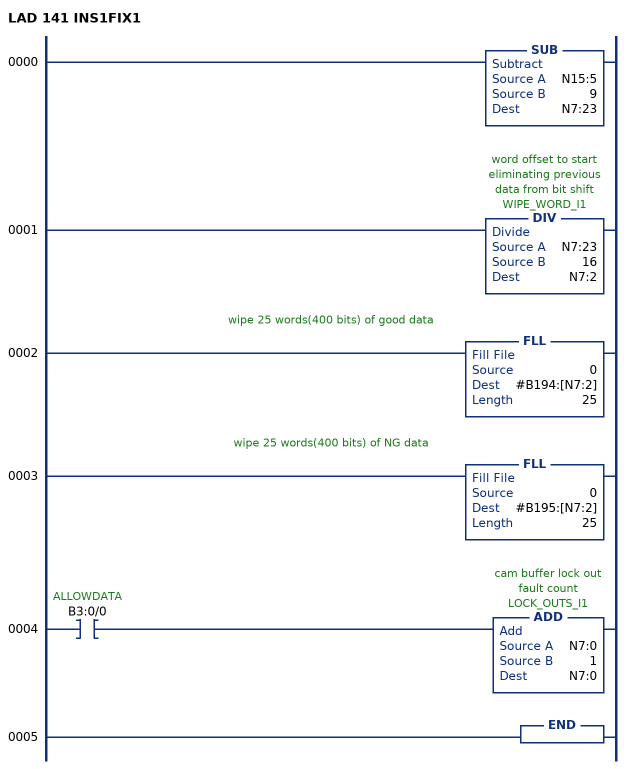
% Rung: 0 %
SOR SUB N15:5 9 N7:23 EOR
%   N15:5  INS_1_TRIG_LOC %
% Rung: 1 %
SOR DIV N7:23 16 N7:2 EOR
%   N7:2  WIPE_WORD_I1  "word offset to start eliminating previous data from bit shift" %
% Rung: 2 %
% wipe 25 words(400 bits) of good data %
SOR FLL 0 #B194:[N7:2] 25 EOR
%   N7:2  WIPE_WORD_I1  "word offset to start eliminating previous data from bit shift" %
% Rung: 3 %
% wipe 25 words(400 bits) of NG data %
SOR FLL 0 #B195:[N7:2] 25 EOR
%   N7:2  WIPE_WORD_I1  "word offset to start eliminating previous data from bit shift" %
% Rung: 4 %
SOR XIC B3:0/0 ADD N7:0 1 N7:0 EOR
%   B3:0/0  ALLOWDATA %
%   N7:0  LOCK_OUTS_I1  "cam buffer lock out fault count" %
% Rung: 5 %
SOR END EOR

LADDER 142 "INS1FIX2"
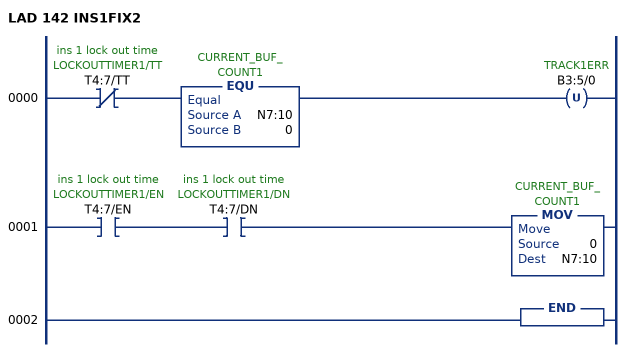
% Rung: 0 %
SOR XIO T4:7/TT EQU N7:10 0 OTU B3:5/0 EOR
%   T4:7  LOCKOUTTIMER1  "ins 1 lock out time" %
%   N7:10  CURRENT_BUF_COUNT1 %
%   B3:5/0  TRACK1ERR %
% Rung: 1 %
SOR XIC T4:7/EN XIC T4:7/DN MOV 0 N7:10 EOR
%   T4:7  LOCKOUTTIMER1  "ins 1 lock out time" %
%   N7:10  CURRENT_BUF_COUNT1 %
% Rung: 2 %
SOR END EOR

LADDER 145 "INS2"
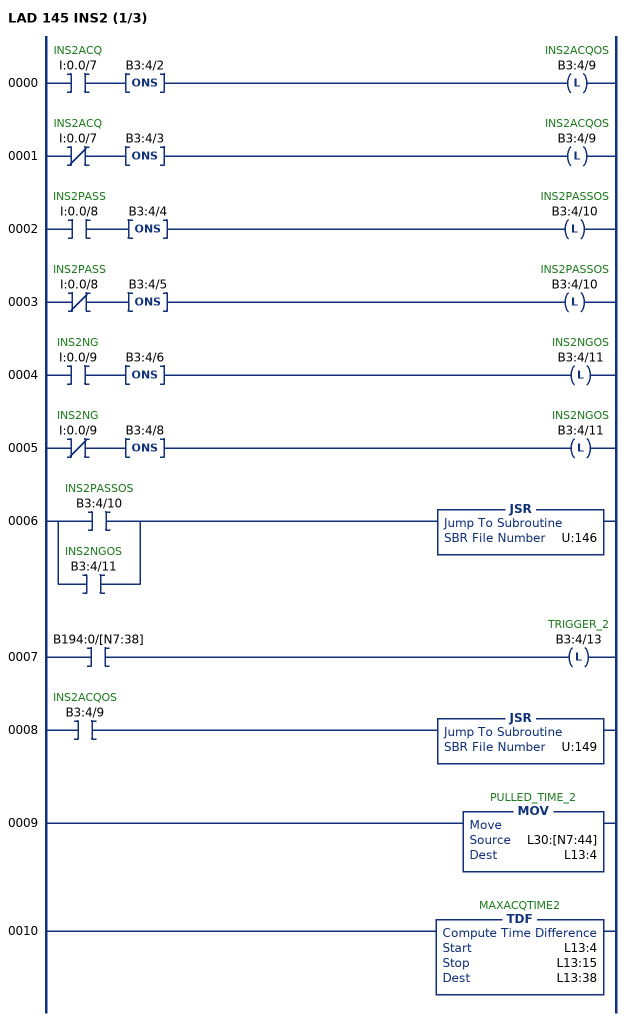
% Rung: 0 %
SOR XIC I:0.0/7 ONS B3:4/2 OTL B3:4/9 EOR
%   I:0.0/7  INS2ACQ %
%   B3:4/9  INS2ACQOS %
% Rung: 1 %
SOR XIO I:0.0/7 ONS B3:4/3 OTL B3:4/9 EOR
%   I:0.0/7  INS2ACQ %
%   B3:4/9  INS2ACQOS %
% Rung: 2 %
SOR XIC I:0.0/8 ONS B3:4/4 OTL B3:4/10 EOR
%   I:0.0/8  INS2PASS %
%   B3:4/10  INS2PASSOS %
% Rung: 3 %
SOR XIO I:0.0/8 ONS B3:4/5 OTL B3:4/10 EOR
%   I:0.0/8  INS2PASS %
%   B3:4/10  INS2PASSOS %
% Rung: 4 %
SOR XIC I:0.0/9 ONS B3:4/6 OTL B3:4/11 EOR
%   I:0.0/9  INS2NG %
%   B3:4/11  INS2NGOS %
% Rung: 5 %
SOR XIO I:0.0/9 ONS B3:4/8 OTL B3:4/11 EOR
%   I:0.0/9  INS2NG %
%   B3:4/11  INS2NGOS %
% Rung: 6 %
SOR BST XIC B3:4/10 NXB XIC B3:4/11 BND JSR U:146 EOR
%   B3:4/10  INS2PASSOS %
%   B3:4/11  INS2NGOS %
% Rung: 7 %
SOR XIC B194:0/[N7:38] OTL B3:4/13 EOR
%   B194:0  BOT_GOOD_FILE %
%   N7:38  INS_2_TRIG_LOC %
%   B3:4/13  TRIGGER_2 %
% Rung: 8 %
SOR XIC B3:4/9 JSR U:149 EOR
%   B3:4/9  INS2ACQOS %
% Rung: 9 %
SOR MOV L30:[N7:44] L13:4 EOR
%   N7:44  OLDEST_PART_INDEX2 %
%   L13:4  PULLED_TIME_2 %
% Rung: 10 %
SOR TDF L13:4 L13:15 L13:38 EOR
%   L13:4  PULLED_TIME_2 %
%   L13:15  BOT_TIME %
%   L13:38  MAXACQTIME2 %

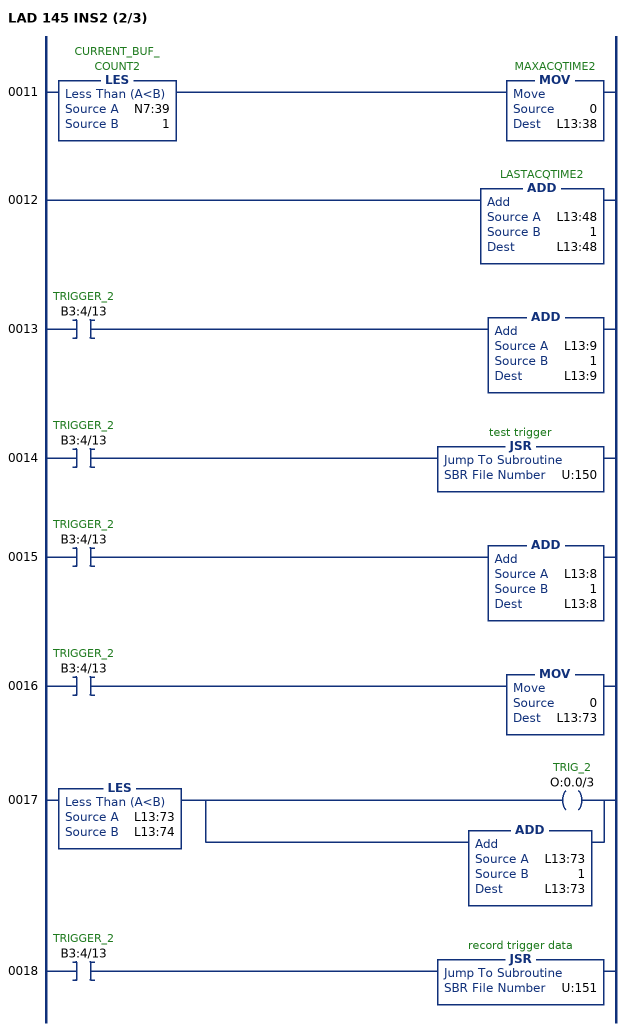
% Rung: 11 %
SOR LES N7:39 1 MOV 0 L13:38 EOR
%   N7:39  CURRENT_BUF_COUNT2 %
%   L13:38  MAXACQTIME2 %
% Rung: 12 %
SOR ADD L13:48 1 L13:48 EOR
%   L13:48  LASTACQTIME2 %
% Rung: 13 %
SOR XIC B3:4/13 ADD L13:9 1 L13:9 EOR
%   B3:4/13  TRIGGER_2 %
% Rung: 14 %
SOR XIC B3:4/13 JSR U:150 EOR
%   B3:4/13  TRIGGER_2 %
%   U:150  "test trigger" %
% Rung: 15 %
SOR XIC B3:4/13 ADD L13:8 1 L13:8 EOR
%   B3:4/13  TRIGGER_2 %
% Rung: 16 %
SOR XIC B3:4/13 MOV 0 L13:73 EOR
%   B3:4/13  TRIGGER_2 %
% Rung: 17 %
SOR LES L13:73 L13:74 BST OTE O:0.0/3 NXB ADD L13:73 1 L13:73 BND EOR
%   O:0.0/3  TRIG_2 %
% Rung: 18 %
SOR XIC B3:4/13 JSR U:151 EOR
%   B3:4/13  TRIGGER_2 %
%   U:151  "record trigger data" %

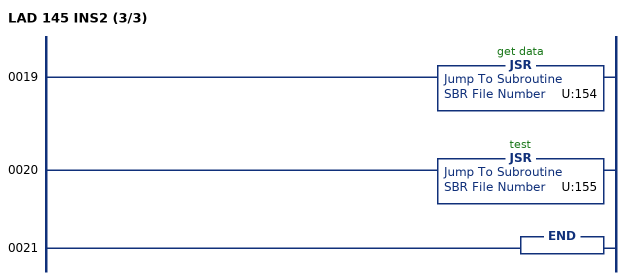
% Rung: 19 %
SOR JSR U:154 EOR
%   U:154  "get data" %
% Rung: 20 %
SOR JSR U:155 EOR
%   U:155  "test" %
% Rung: 21 %
SOR END EOR

LADDER 146 "INS2RESULT"
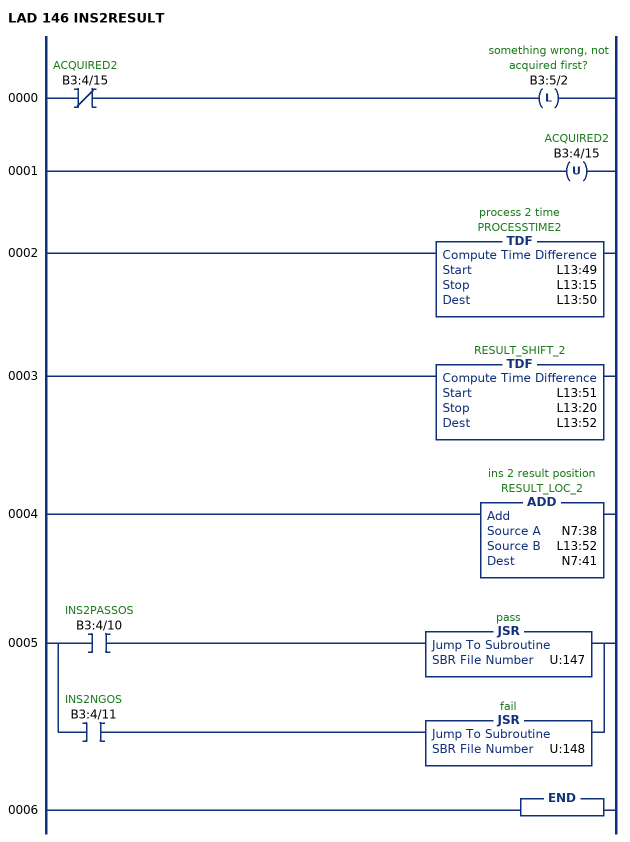
% Rung: 0 %
SOR XIO B3:4/15 OTL B3:5/2 EOR
%   B3:4/15  ACQUIRED2 %
%   B3:5/2  "something wrong, not acquired first?" %
% Rung: 1 %
SOR OTU B3:4/15 EOR
%   B3:4/15  ACQUIRED2 %
% Rung: 2 %
SOR TDF L13:49 L13:15 L13:50 EOR
%   L13:49  TIMEOFACQ2  "the time of the last acquire" %
%   L13:15  BOT_TIME %
%   L13:50  PROCESSTIME2  "process 2 time" %
% Rung: 3 %
SOR TDF L13:51 L13:20 L13:52 EOR
%   L13:51  PROCESS_START_POS_2 %
%   L13:20  BOT_POSITION %
%   L13:52  RESULT_SHIFT_2 %
% Rung: 4 %
SOR ADD N7:38 L13:52 N7:41 EOR
%   N7:38  INS_2_TRIG_LOC %
%   L13:52  RESULT_SHIFT_2 %
%   N7:41  RESULT_LOC_2  "ins 2 result position" %
% Rung: 5 %
SOR BST XIC B3:4/10 JSR U:147 NXB XIC B3:4/11 JSR U:148 BND EOR
%   B3:4/10  INS2PASSOS %
%   U:147  "pass" %
%   B3:4/11  INS2NGOS %
%   U:148  "fail" %
% Rung: 6 %
SOR END EOR

LADDER 147 "INS2PASS"
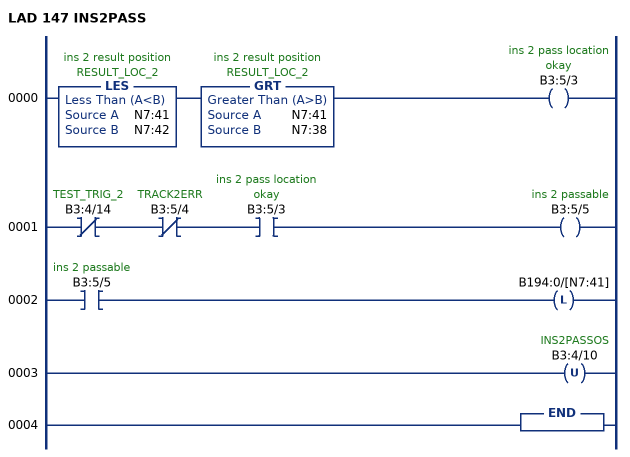
% Rung: 0 %
SOR LES N7:41 N7:42 GRT N7:41 N7:38 OTE B3:5/3 EOR
%   N7:41  RESULT_LOC_2  "ins 2 result position" %
%   N7:42  MAXRSTLOC2 %
%   N7:38  INS_2_TRIG_LOC %
%   B3:5/3  "ins 2 pass location okay" %
% Rung: 1 %
SOR XIO B3:4/14 XIO B3:5/4 XIC B3:5/3 OTE B3:5/5 EOR
%   B3:4/14  TEST_TRIG_2 %
%   B3:5/4  TRACK2ERR %
%   B3:5/3  "ins 2 pass location okay" %
%   B3:5/5  "ins 2 passable" %
% Rung: 2 %
SOR XIC B3:5/5 OTL B194:0/[N7:41] EOR
%   B3:5/5  "ins 2 passable" %
%   B194:0  BOT_GOOD_FILE %
%   N7:41  RESULT_LOC_2  "ins 2 result position" %
% Rung: 3 %
SOR OTU B3:4/10 EOR
%   B3:4/10  INS2PASSOS %
% Rung: 4 %
SOR END EOR

LADDER 148 "INS2FAIL"
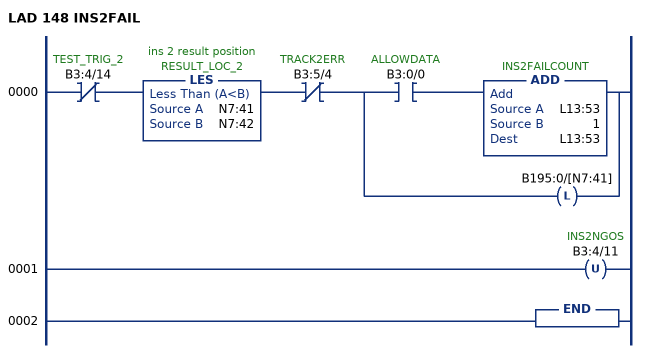
% Rung: 0 %
SOR XIO B3:4/14 LES N7:41 N7:42 XIO B3:5/4 BST XIC B3:0/0 ADD L13:53 1 L13:53 NXB OTL B195:0/[N7:41] BND EOR
%   B3:4/14  TEST_TRIG_2 %
%   N7:41  RESULT_LOC_2  "ins 2 result position" %
%   N7:42  MAXRSTLOC2 %
%   B3:5/4  TRACK2ERR %
%   B3:0/0  ALLOWDATA %
%   L13:53  INS2FAILCOUNT %
%   B195:0  BOT_NG_FILE %
% Rung: 1 %
SOR OTU B3:4/11 EOR
%   B3:4/11  INS2NGOS %
% Rung: 2 %
SOR END EOR

LADDER 149 "INS2ACQ"
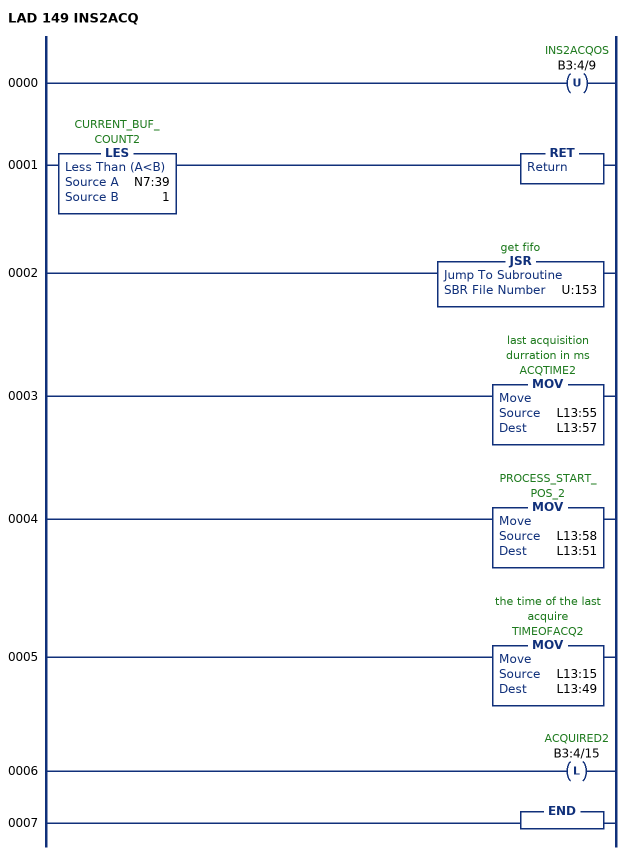
% Rung: 0 %
SOR OTU B3:4/9 EOR
%   B3:4/9  INS2ACQOS %
% Rung: 1 %
SOR LES N7:39 1 RET EOR
%   N7:39  CURRENT_BUF_COUNT2 %
% Rung: 2 %
SOR JSR U:153 EOR
%   U:153  "get fifo" %
% Rung: 3 %
SOR MOV L13:55 L13:57 EOR
%   L13:55  TIME_SPAN2 %
%   L13:57  ACQTIME2  "last acquisition durration in ms" %
% Rung: 4 %
SOR MOV L13:58 L13:51 EOR
%   L13:58  PULLED_POSITION2 %
%   L13:51  PROCESS_START_POS_2 %
% Rung: 5 %
SOR MOV L13:15 L13:49 EOR
%   L13:15  BOT_TIME %
%   L13:49  TIMEOFACQ2  "the time of the last acquire" %
% Rung: 6 %
SOR OTL B3:4/15 EOR
%   B3:4/15  ACQUIRED2 %
% Rung: 7 %
SOR END EOR

LADDER 150 "Q2TIMETEST"
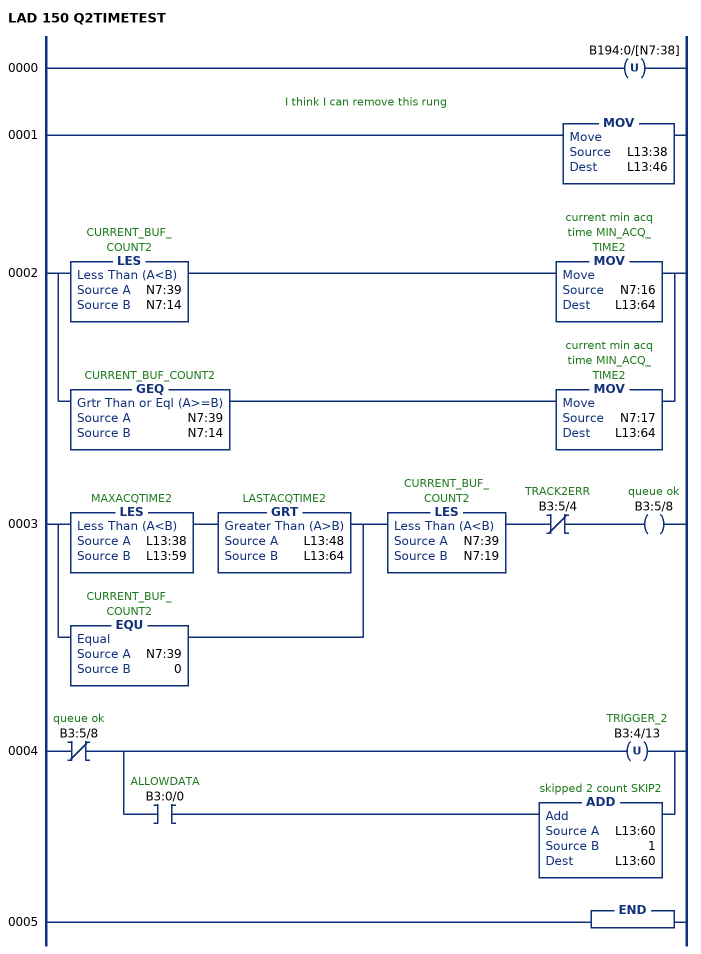
% Rung: 0 %
SOR OTU B194:0/[N7:38] EOR
%   B194:0  BOT_GOOD_FILE %
%   N7:38  INS_2_TRIG_LOC %
% Rung: 1 %
% I think I can remove this rung %
SOR MOV L13:38 L13:46 EOR
%   L13:38  MAXACQTIME2 %
% Rung: 2 %
SOR BST LES N7:39 N7:14 MOV N7:16 L13:64 NXB GEQ N7:39 N7:14 MOV N7:17 L13:64 BND EOR
%   N7:39  CURRENT_BUF_COUNT2 %
%   N7:14  "Max high speed buffers" %
%   N7:16  "high speed acquisition time" %
%   L13:64  MIN_ACQ_TIME2  "current min acq time" %
%   N7:17  "low speed acquisition time" %
% Rung: 3 %
SOR BST LES L13:38 L13:59 GRT L13:48 L13:64 NXB EQU N7:39 0 BND LES N7:39 N7:19 XIO B3:5/4 OTE B3:5/8 EOR
%   L13:38  MAXACQTIME2 %
%   L13:59  ACQTIMELIMIT2 %
%   L13:48  LASTACQTIME2 %
%   L13:64  MIN_ACQ_TIME2  "current min acq time" %
%   N7:39  CURRENT_BUF_COUNT2 %
%   N7:19  MAX_BUFF  "maximum buffers" %
%   B3:5/4  TRACK2ERR %
%   B3:5/8  "queue ok" %
% Rung: 4 %
SOR XIO B3:5/8 BST OTU B3:4/13 NXB XIC B3:0/0 ADD L13:60 1 L13:60 BND EOR
%   B3:5/8  "queue ok" %
%   B3:4/13  TRIGGER_2 %
%   B3:0/0  ALLOWDATA %
%   L13:60  SKIP2  "skipped 2 count" %
% Rung: 5 %
SOR END EOR

LADDER 151 "INS2TRIG"
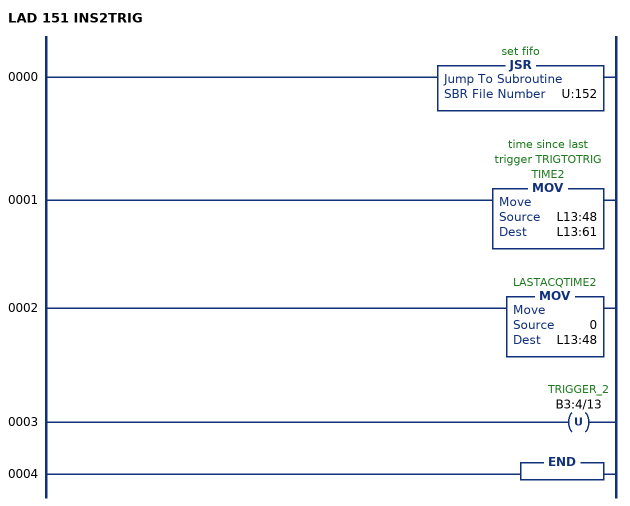
% Rung: 0 %
SOR JSR U:152 EOR
%   U:152  "set fifo" %
% Rung: 1 %
SOR MOV L13:48 L13:61 EOR
%   L13:48  LASTACQTIME2 %
%   L13:61  TRIGTOTRIGTIME2  "time since last trigger" %
% Rung: 2 %
SOR MOV 0 L13:48 EOR
%   L13:48  LASTACQTIME2 %
% Rung: 3 %
SOR OTU B3:4/13 EOR
%   B3:4/13  TRIGGER_2 %
% Rung: 4 %
SOR END EOR

LADDER 152 "FIFO2SET"
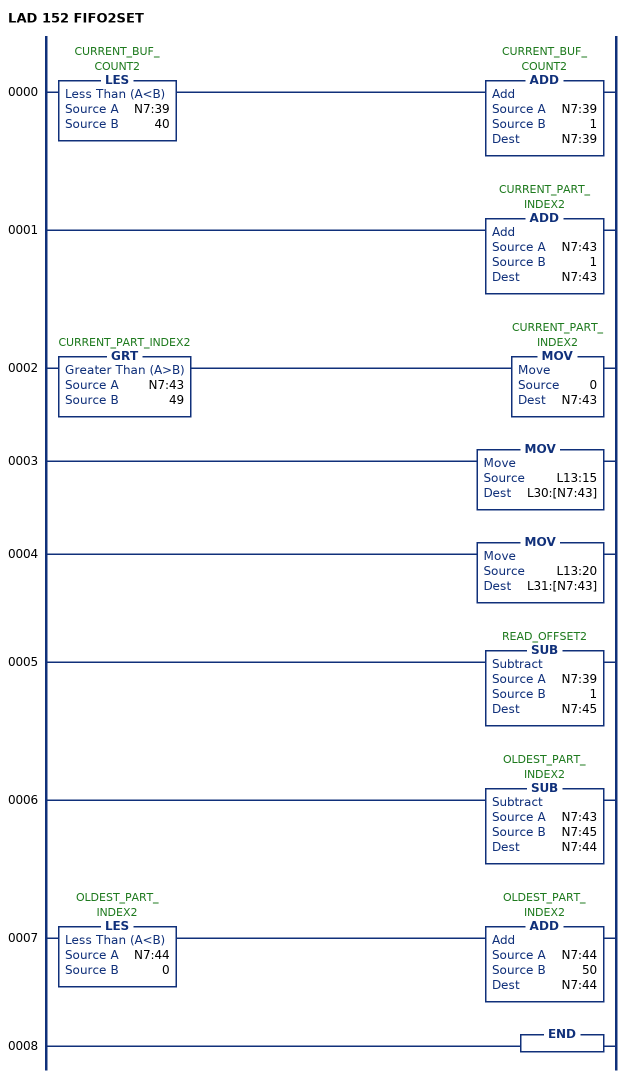
% Rung: 0 %
SOR LES N7:39 40 ADD N7:39 1 N7:39 EOR
%   N7:39  CURRENT_BUF_COUNT2 %
% Rung: 1 %
SOR ADD N7:43 1 N7:43 EOR
%   N7:43  CURRENT_PART_INDEX2 %
% Rung: 2 %
SOR GRT N7:43 49 MOV 0 N7:43 EOR
%   N7:43  CURRENT_PART_INDEX2 %
% Rung: 3 %
SOR MOV L13:15 L30:[N7:43] EOR
%   L13:15  BOT_TIME %
%   N7:43  CURRENT_PART_INDEX2 %
% Rung: 4 %
SOR MOV L13:20 L31:[N7:43] EOR
%   L13:20  BOT_POSITION %
%   N7:43  CURRENT_PART_INDEX2 %
% Rung: 5 %
SOR SUB N7:39 1 N7:45 EOR
%   N7:39  CURRENT_BUF_COUNT2 %
%   N7:45  READ_OFFSET2 %
% Rung: 6 %
SOR SUB N7:43 N7:45 N7:44 EOR
%   N7:43  CURRENT_PART_INDEX2 %
%   N7:45  READ_OFFSET2 %
%   N7:44  OLDEST_PART_INDEX2 %
% Rung: 7 %
SOR LES N7:44 0 ADD N7:44 50 N7:44 EOR
%   N7:44  OLDEST_PART_INDEX2 %
% Rung: 8 %
SOR END EOR

LADDER 153 "FIFO2GET"
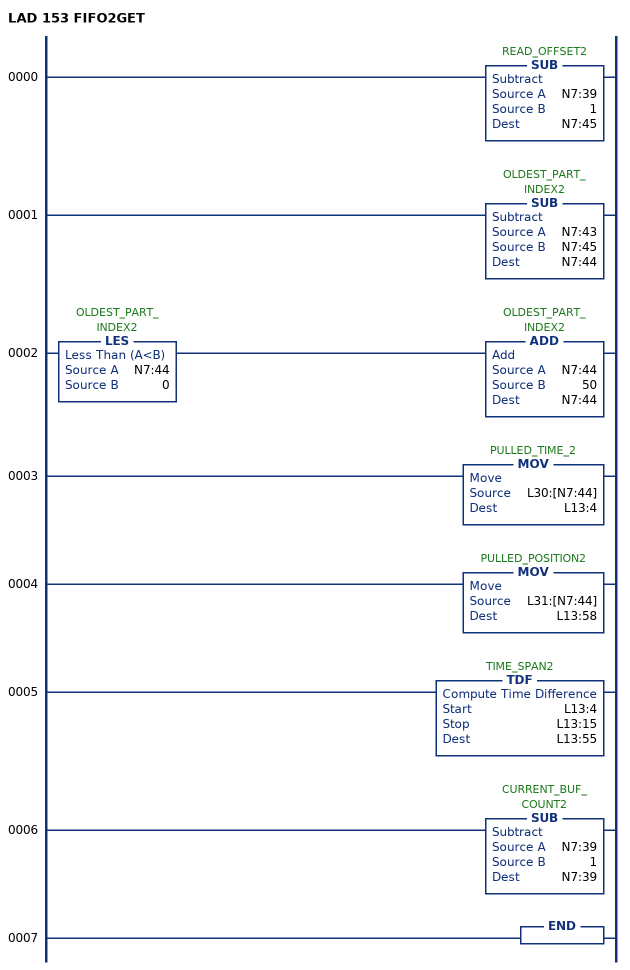
% Rung: 0 %
SOR SUB N7:39 1 N7:45 EOR
%   N7:39  CURRENT_BUF_COUNT2 %
%   N7:45  READ_OFFSET2 %
% Rung: 1 %
SOR SUB N7:43 N7:45 N7:44 EOR
%   N7:43  CURRENT_PART_INDEX2 %
%   N7:45  READ_OFFSET2 %
%   N7:44  OLDEST_PART_INDEX2 %
% Rung: 2 %
SOR LES N7:44 0 ADD N7:44 50 N7:44 EOR
%   N7:44  OLDEST_PART_INDEX2 %
% Rung: 3 %
SOR MOV L30:[N7:44] L13:4 EOR
%   N7:44  OLDEST_PART_INDEX2 %
%   L13:4  PULLED_TIME_2 %
% Rung: 4 %
SOR MOV L31:[N7:44] L13:58 EOR
%   N7:44  OLDEST_PART_INDEX2 %
%   L13:58  PULLED_POSITION2 %
% Rung: 5 %
SOR TDF L13:4 L13:15 L13:55 EOR
%   L13:4  PULLED_TIME_2 %
%   L13:15  BOT_TIME %
%   L13:55  TIME_SPAN2 %
% Rung: 6 %
SOR SUB N7:39 1 N7:39 EOR
%   N7:39  CURRENT_BUF_COUNT2 %
% Rung: 7 %
SOR END EOR

LADDER 154 "INSDATA2"    % used for analysis %
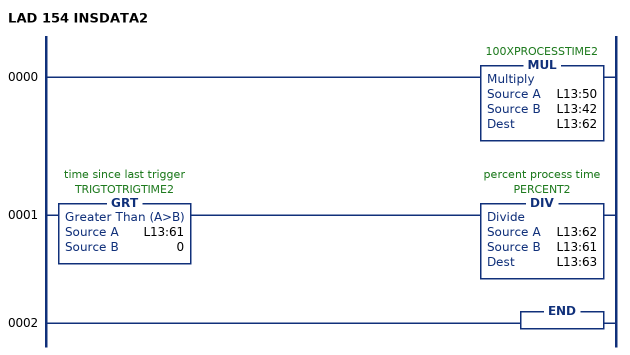
% Rung: 0 %
SOR MUL L13:50 L13:42 L13:62 EOR
%   L13:50  PROCESSTIME2  "process 2 time" %
%   L13:42  100X_MULTIPLIER %
%   L13:62  100XPROCESSTIME2 %
% Rung: 1 %
SOR GRT L13:61 0 DIV L13:62 L13:61 L13:63 EOR
%   L13:61  TRIGTOTRIGTIME2  "time since last trigger" %
%   L13:62  100XPROCESSTIME2 %
%   L13:63  PERCENT2  "percent process time" %
% Rung: 2 %
SOR END EOR

LADDER 155 "TESTFAULT2"
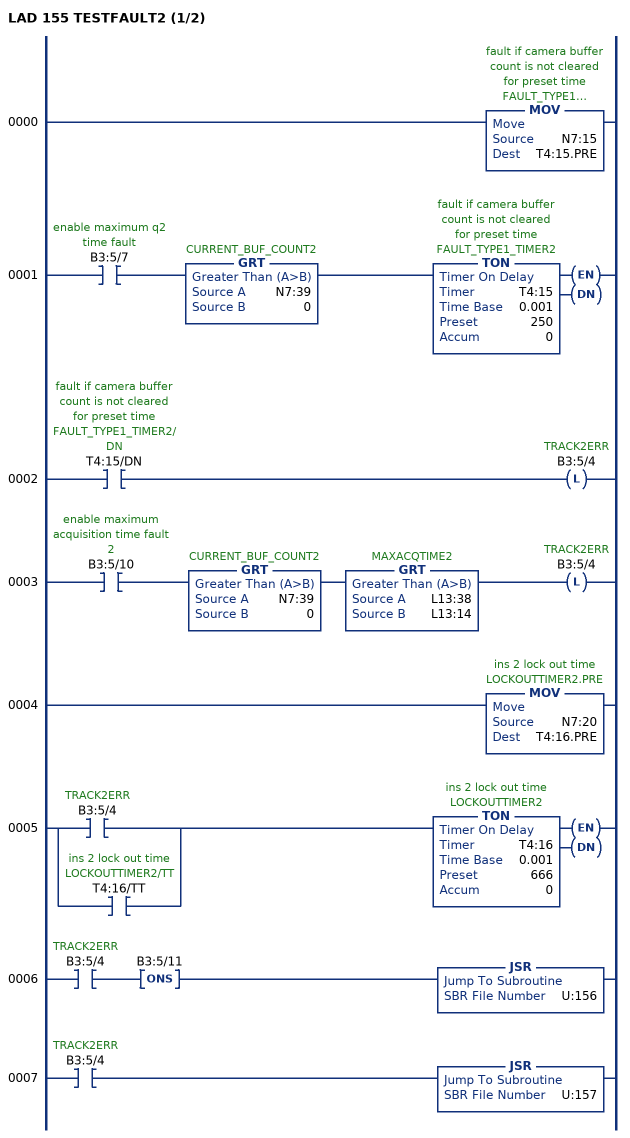
% Rung: 0 %
SOR MOV N7:15 T4:15.PRE EOR
%   N7:15  MAXQ1TMFLT  "max allowed ms time for q to be above 1 if safe fault is used" %
%   T4:15  FAULT_TYPE1_TIMER2  "fault if camera buffer count is not cleared for preset time" %
% Rung: 1 %
SOR XIC B3:5/7 GRT N7:39 0 TON T4:15 0.001 250 0 EOR
%   B3:5/7  "enable maximum q2 time fault" %
%   N7:39  CURRENT_BUF_COUNT2 %
%   T4:15  FAULT_TYPE1_TIMER2  "fault if camera buffer count is not cleared for preset time" %
% Rung: 2 %
SOR XIC T4:15/DN OTL B3:5/4 EOR
%   T4:15  FAULT_TYPE1_TIMER2  "fault if camera buffer count is not cleared for preset time" %
%   B3:5/4  TRACK2ERR %
% Rung: 3 %
SOR XIC B3:5/10 GRT N7:39 0 GRT L13:38 L13:14 OTL B3:5/4 EOR
%   B3:5/10  "enable maximum acquisition time fault 2" %
%   N7:39  CURRENT_BUF_COUNT2 %
%   L13:38  MAXACQTIME2 %
%   L13:14  LONGESTACQUIRETIME  "maximum of the longest acquire time allowed if maximum acquire time fault is enabled" %
%   B3:5/4  TRACK2ERR %
% Rung: 4 %
SOR MOV N7:20 T4:16.PRE EOR
%   N7:20  LOCKOUTTIME  "ms time setting to lock out inspection to give all pending images a chance to clear" %
%   T4:16  LOCKOUTTIMER2  "ins 2 lock out time" %
% Rung: 5 %
SOR BST XIC B3:5/4 NXB XIC T4:16/TT BND TON T4:16 0.001 666 0 EOR
%   B3:5/4  TRACK2ERR %
%   T4:16  LOCKOUTTIMER2  "ins 2 lock out time" %
% Rung: 6 %
SOR XIC B3:5/4 ONS B3:5/11 JSR U:156 EOR
%   B3:5/4  TRACK2ERR %
% Rung: 7 %
SOR XIC B3:5/4 JSR U:157 EOR
%   B3:5/4  TRACK2ERR %

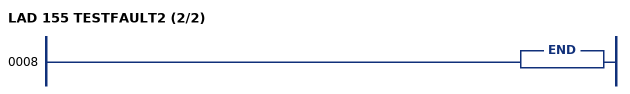
% Rung: 8 %
SOR END EOR

LADDER 156 "INS2FIX1"
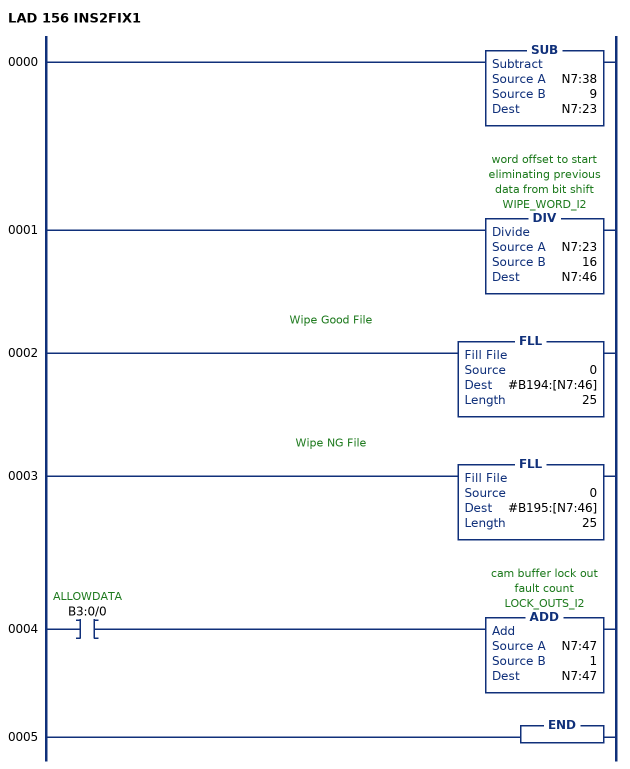
% Rung: 0 %
SOR SUB N7:38 9 N7:23 EOR
%   N7:38  INS_2_TRIG_LOC %
% Rung: 1 %
SOR DIV N7:23 16 N7:46 EOR
%   N7:46  WIPE_WORD_I2  "word offset to start eliminating previous data from bit shift" %
% Rung: 2 %
% Wipe Good File %
SOR FLL 0 #B194:[N7:46] 25 EOR
%   N7:46  WIPE_WORD_I2  "word offset to start eliminating previous data from bit shift" %
% Rung: 3 %
% Wipe NG File %
SOR FLL 0 #B195:[N7:46] 25 EOR
%   N7:46  WIPE_WORD_I2  "word offset to start eliminating previous data from bit shift" %
% Rung: 4 %
SOR XIC B3:0/0 ADD N7:47 1 N7:47 EOR
%   B3:0/0  ALLOWDATA %
%   N7:47  LOCK_OUTS_I2  "cam buffer lock out fault count" %
% Rung: 5 %
SOR END EOR

LADDER 157 "INS2FIX2"
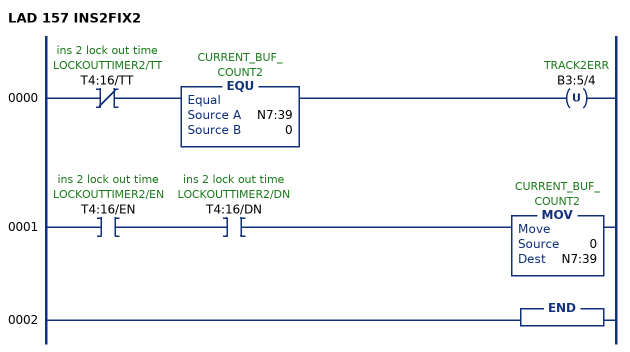
% Rung: 0 %
SOR XIO T4:16/TT EQU N7:39 0 OTU B3:5/4 EOR
%   T4:16  LOCKOUTTIMER2  "ins 2 lock out time" %
%   N7:39  CURRENT_BUF_COUNT2 %
%   B3:5/4  TRACK2ERR %
% Rung: 1 %
SOR XIC T4:16/EN XIC T4:16/DN MOV 0 N7:39 EOR
%   T4:16  LOCKOUTTIMER2  "ins 2 lock out time" %
%   N7:39  CURRENT_BUF_COUNT2 %
% Rung: 2 %
SOR END EOR

LADDER 200 "XFEROUT"
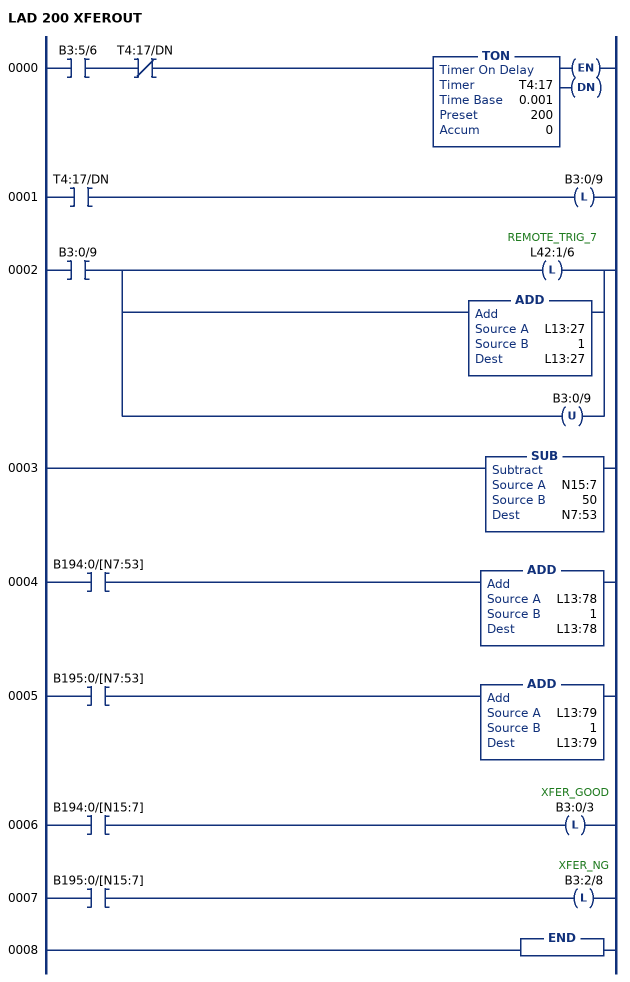
% Rung: 0 %
SOR XIC B3:5/6 XIO T4:17/DN TON T4:17 0.001 200 0 EOR
% Rung: 1 %
SOR XIC T4:17/DN OTL B3:0/9 EOR
% Rung: 2 %
SOR XIC B3:0/9 BST OTL L42:1/6 NXB ADD L13:27 1 L13:27 NXB OTU B3:0/9 BND EOR
%   L42:1/6  REMOTE_TRIG_7 %
% Rung: 3 %
SOR SUB N15:7 50 N7:53 EOR
%   N15:7  XFER_OUT_LOC %
% Rung: 4 %
SOR XIC B194:0/[N7:53] ADD L13:78 1 L13:78 EOR
%   B194:0  BOT_GOOD_FILE %
% Rung: 5 %
SOR XIC B195:0/[N7:53] ADD L13:79 1 L13:79 EOR
%   B195:0  BOT_NG_FILE %
% Rung: 6 %
SOR XIC B194:0/[N15:7] OTL B3:0/3 EOR
%   B194:0  BOT_GOOD_FILE %
%   N15:7  XFER_OUT_LOC %
%   B3:0/3  XFER_GOOD %
% Rung: 7 %
SOR XIC B195:0/[N15:7] OTL B3:2/8 EOR
%   B195:0  BOT_NG_FILE %
%   N15:7  XFER_OUT_LOC %
%   B3:2/8  XFER_NG %
% Rung: 8 %
SOR END EOR

LADDER 201 "XFER GOOD"
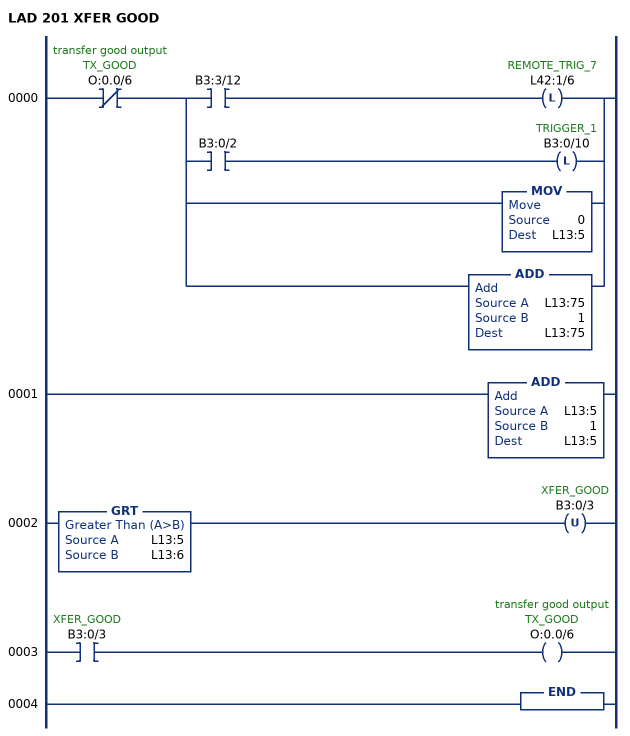
% Rung: 0 %
SOR XIO O:0.0/6 BST XIC B3:3/12 OTL L42:1/6 NXB XIC B3:0/2 OTL B3:0/10 NXB MOV 0 L13:5 NXB ADD L13:75 1 L13:75 BND EOR
%   O:0.0/6  TX_GOOD  "transfer good output" %
%   L42:1/6  REMOTE_TRIG_7 %
%   B3:0/10  TRIGGER_1 %
% Rung: 1 %
SOR ADD L13:5 1 L13:5 EOR
% Rung: 2 %
SOR GRT L13:5 L13:6 OTU B3:0/3 EOR
%   B3:0/3  XFER_GOOD %
% Rung: 3 %
SOR XIC B3:0/3 OTE O:0.0/6 EOR
%   B3:0/3  XFER_GOOD %
%   O:0.0/6  TX_GOOD  "transfer good output" %
% Rung: 4 %
SOR END EOR

LADDER 202 "XFER NG"
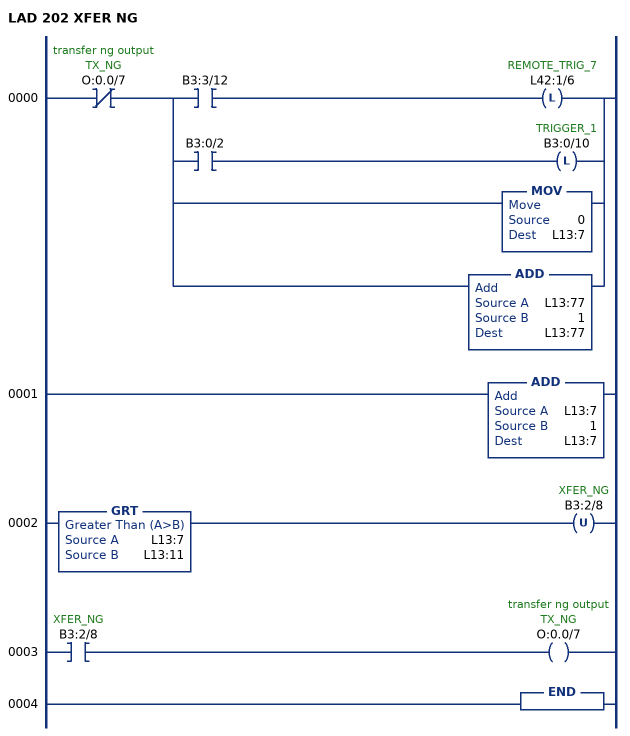
% Rung: 0 %
SOR XIO O:0.0/7 BST XIC B3:3/12 OTL L42:1/6 NXB XIC B3:0/2 OTL B3:0/10 NXB MOV 0 L13:7 NXB ADD L13:77 1 L13:77 BND EOR
%   O:0.0/7  TX_NG  "transfer ng output" %
%   L42:1/6  REMOTE_TRIG_7 %
%   B3:0/10  TRIGGER_1 %
% Rung: 1 %
SOR ADD L13:7 1 L13:7 EOR
% Rung: 2 %
SOR GRT L13:7 L13:11 OTU B3:2/8 EOR
%   B3:2/8  XFER_NG %
% Rung: 3 %
SOR XIC B3:2/8 OTE O:0.0/7 EOR
%   B3:2/8  XFER_NG %
%   O:0.0/7  TX_NG  "transfer ng output" %
% Rung: 4 %
SOR END EOR

OTHER DOCUMENTED ADDRESSES
  B3:5/9  "test for fault conditions"
  B3:5/12  "enable test trigger 2 high speed logic"
  B3:7/5  "enable test trigger 1 high speed logic"
  B196:0/0  "toggle"
  F8:12  "air pressure as float for hmi"
  F8:98  "time in multiples of 10 us"
  F8:99  "loop time in milliseconds"
  F14:3  TOP_SPD_SETPOINT
  I:0.0/0  BOTENCA
  I:0.0/1  BOTENCB
  I:2.0/3  FRONT_ESTOP
  I:2.0/4  REAR_ESTOP
  I:2.0/5  FRONT_DOORS
  I:2.0/6  REAR_DOORS
  I:2.0/10  "spare"
  I:2.0/12  "spare"
  I:2.0/14  "spare"
  L13:54  "test fire interval"
  L13:88  "test fire count index"
  L13:89  "test fire count"
  L13:91  "test fire interval index"
  L42:0/1  "ps stop read (unused)"
  L42:0/3  "bottom enable read (unused)"
  L42:1/2  "box full write (unused)"
  N7:5  NEXT_TIME_INDEX
  N7:6  OLDEST_TIME_INDEX
  N7:7  RATE_PART_COUNT
  N7:8  THIS_TIME_INDEX
  N7:9  UPPER_INDEX_LIMIT
  O:0.0/1  "spare? chute sensor?"
  O:0.0/4  TRIG_3  "spare"
  O:0.0/5  TRIG_4  "spare"
  O:0.0/9  "spare"
  O:0.0/10  "spare"
  O:0.0/11  "spare"
  O:3.0/0  "spare"
  O:3.0/2  "spare"
  O:3.0/3  LT_CTRN_RANGE_SELECT
  O:3.0/8  "spare"
  O:3.0/9  "spare"
  PFILE:6  "check for part jams"
  PFILE:10  "Bottom belt HSC"
  PFILE:12  "Top belt HSC"
  PFILE:123  "used for annylsys"
  Q2:55  END_OF_MAIN
  U:222  "add a part information for rate calculation"
  U:223  "update the rate value"

COMMENTS NOT ATTACHED TO A CURRENT RUNG
  N17:8: ****************************************************************************************************************
    I can not find anywhere in the program where the "Test Spacing From Pickup to Trigger is activated indicating to me that this entire function must not be doing anything in this program at this time.
    ****************************************************************************************************************
  T20:2: The timer used to verify that the part that triggered the top laser optic has passed the bottom camer. needs to be count
  T20:2.ACC: This rung is starting a timer that should be activated directly before the laser optic part presense sensor on the top conveyer and should cause the top optic to be ignored if the bottom camera system didn't pass. however other arrangements must be made if the bottom camera isn't going to be used as is the case with a nut inspection.
  B22:0/0: ***********************
     Bottom Part Syncronizing Logic
    ***********************
    
    This is the point at the bottom of the top conveyor where the part jumps from the bottom conveyor.  This system will then track the part through the top system to the point of the laser optic in order to verify that the part in question has passed the bottom inspection.  I believe that we NEED to include FAILING inspections to eliminate the possibility of a out of position part from passing. LW 072010
  C5:4: tempory counting to verify pass part count with boxing part count.
  B23:0/0: Yet another bit shift load with data in the part position indicating that there was a bottom system part pass as well as a top system part present at this location.
    
    verified works w/bypassed 071910 and unbypassed 072010
  I:0.0/8: special rung for testing. This rung can simulate a pass signal. It will not be timed correctly.
  F8:13: *************************
    Loads Side Camera Passing data into a bit shift
    *************************
    
    loads passing data bit into passing data bit shift register at the part present cl.
  B3:7/9: ************************************
     The next 3 rungs appear to do nothing
    ***********************************
  B11:0/0: load part present bit shit with one shot data from the part present sensor
  RUNG000127-000009: multiply the current image acquire q by 11(ms) to get the current skip trigger delay
  RUNG000127-000010: time since oldest trigger
  RUNG000127-000012: trigger / capture part at trigger location
  RUNG000127-000015: time since last trigger
  RUNG000127-000017: remove used trigger bit
  B3:6/1: ***********************
    Part Width and  Location
    ***********************
    
    Calculates the position of parts on the top belt by measureing the part width by calculating the number of belt movement pulses that occure when the optic is blocked and then devides that in half and add that to the optic location in the part presnet bit shift when the top optic is cleared.
  B3:6/0: make a bit come on indicating that a part that passed the bottom camera is within  range when crossing the top camera.
  B9:0/[N7:47]: Remove any part present signals outside of expected location
  B9:0/[N7:50]: Remove any part present signals outside of expected location
  F19:0: Counter inside of a high speed counter interrupt counts the number of Bit Shifts that need to be processed in order to move the logic with the parts on the conveyor.
  F8:14: **************
    Bottom Top Camera Trigger
    *************
    
    Trigger Bottom Top Camera
  L13:104: Tracking error handler
  N10:4: test if boxing is connected
  T4:28: Check for buffer reset
  B3:11/3: After initial delay allow blow two start functioning
  RUNG000150-000041: transfer tracked part positon from trigger/acquire to the acquire/result
    capture acquire time
    reset process time
  RUNG000150-000039: Grab trigger/acquire position
    Grab acquire time
  RUNG000150-000038: acquire code
  RUNG000150-000035: fail count
  RUNG000150-000032: pass count
  RUNG000150-000025: pass code / Set pass bit in Bit Shift
    captures result position and processing time
    Unlatch pass bit
  RUNG000150-000018: pass, fail and acquire inputs
  RUNG000150-000016: wiped count
  RUNG000150-000014: clear data for time
  RUNG000150-000013: clear data for aquire time expired
  RUNG000150-000012: wipe stored part data if acq time expires
  RUNG000150-000011: trigger count
  L13:101: record the minimum time between triggers
  L14:5: on when ok to run, rear off turns both off
  L14:2: off when ok to run
  L14:3: off when ok to run
  L14:8: on when ok for run
  N7:76: removed relieance on trigger signal
  N197:20/0: Passes deformed head blowoff command to TOP PLC where solenoid output is located.
  L13:163: maximum average q
  L13:162: maximum q
  RUNG000141-000007: computer the time difference from the "pulled" data to the current time.
  RUNG000141-000006: convert offset data to a standard data because the TDF function can't handle offsets
  N7:50: ***********************************************************************************************************************************************************
    From top
    ***********************************************************************************************************************************************************
    
    removed relieance on trigger signal
  T4:20: Optic watchdog timers for faults
  B3:10/1: prevents momentary signals from box present sensor from tripping the logic for box not present
    
    This is in responce to a problem created by the sensor occasionally turning on as if no box was in its path when there is a box present.
  B3:6/2: IF PROCESSING FAULT OCURES AT COUNTER SENSOR; CLEAR THE BELT OF PASSING DATA
  L14:36: ****************  nEEDS fIXING  **********************
  L14:23: ****************  nEEDS fIXING  **********************
  RUNG000010-000018: Remove any part present signals outside of expected location
  RUNG000010-000014: ****
                      Zeros out the non passing part count when one passes
    ****
  T4:27: Check for buffer reset
  RUNG000125-000011: trigger count
  RUNG000125-000012: wipe stored part data if acq time expires
  RUNG000125-000013: clear data for aquire time expired
  RUNG000125-000014: clear data for time
  RUNG000125-000016: wiped count
  RUNG000125-000018: pass, fail and acquire inputs
  RUNG000125-000025: pass code / Set pass bit in Bit Shift
    captures result position and processing time
    Unlatch pass bit
  RUNG000125-000026: Grab trigger/acquire position
    Grab acquire time
  RUNG000125-000027: transfer tracked part positon from trigger/acquire to the acquire/result
    capture acquire time
    reset process time
  RUNG000125-000029: Set pass bit in Bit Shift
    captures result position and processing time
    Unlatch pass bit

REVISION NOTES
  13: updated count reset
  14: added io moduals
  15: multiple steps toward new hmi integration
  21: test

DATA TABLE (non-zero values as saved)
DATA B3
% B3:0 % 0X8111 0X1012 0X0061 0XAE80 0X3128 0X0504 0X4602 0X0400 0X4007 0X0000
% B3:10 % 0X2041 0X0846 0X2000 0X0000 0X0000 0X0000 0X0000 0X0000 0X0000 0X0000
DATA T4
% .PRE .ACC %
% T4:0 % 0 1
% T4:1 % 200 0
% T4:2 % 250 154
% T4:3 % 1000 0
% T4:4 % 400 0
% T4:5 % 250 0
% T4:6 % 10 10
% T4:7 % 100 0
% T4:8 % 2 0
% T4:9 % 50 20
% T4:10 % 200 200
% T4:11 % 1 0
% T4:12 % 55 0
% T4:13 % 6 0
% T4:14 % 333 168
% T4:15 % 250 0
% T4:16 % 666 0
% T4:17 % 200 0
% T4:18 % 50 0
% T4:19 % 45 0
% T4:20 % 200 0
% T4:21 % 200 0
% T4:22 % 200 0
% T4:23 % 50 0
% T4:24 % 50 0
% T4:25 % 50 0
% T4:26 % 250 0
% T4:27 % 250 0
% T4:28 % 250 0
% T4:29 % 5000 0
% T4:30 % 50 50
% T4:31 % 20 0
% T4:32 % 69 0
DATA C5
% .PRE .ACC %
% C5:0 % 32766 0
DATA R6
% .LEN .POS %
% R6:0 % 1400 0
% R6:1 % 1400 0
% R6:2 % 1400 0
% R6:3 % 1400 0
% R6:4 % 1400 0
% R6:5 % 1400 0
% R6:6 % 1100 0
% R6:7 % 10 0
% R6:8 % 3 0
% R6:9 % 3 0
% R6:10 % 700 0
% R6:11 % 700 0
% R6:12 % 10 0
% R6:13 % 10 0
% R6:14 % 10 0
% R6:15 % 10 0
% R6:16 % 1100 0
% R6:17 % 700 0
% R6:18 % 700 0
% R6:19 % 10 0
DATA N7
% N7:0 % 1 4 6 1 24574 324 324 501 323 500
% N7:10 % 0 28 0 28 800 250 13 50 32766 9
% N7:20 % 100 333 131 99 250 0 500 600 1000 1600
% N7:30 % 800 100 400 1000 21297 30144 2971 2200 0 0
% N7:40 % 333 7200 1000 30 30 0 57 0 40 47
% N7:50 % 1000 10000 10000 1260 0 1638 18021 0 12 0
% N7:60 % 1 32767 4012 20 31 0 0 15 30 20
% N7:70 % 0 21 23 27738 32767 0 122 0 16 0
% N7:80 % 0 6 95 0 0 0 5 500 0 0
% N7:90 % 2011 4 4 12 1 0 0 0 0 1600
% N7:100 % 1003 90 110 100 175 25 0 0 0 0
DATA F8
% F8:0 % 1 0 0 0 0
% F8:95 % 0 0 0 492 4.92
DATA B9
% B9:130 % 0X0000 0X0000 0X0000 0X0000 0X2000 0X0000 0X0000 0X0000 0X0000 0X8000
% B9:140 % 0X2480 0X0000 0X0000 0X0000 0X0000 0X0000 0X0000 0X0000 0X0000 0X0000
% B9:160 % 0X0000 0X0000 0X0000 0X0000 0X0000 0X0000 0X2000 0X0002 0X0000 0X0000
% B9:170 % 0X0000 0X0000 0X0000 0X2000 0X0000 0X0000 0X0000 0X0000 0X0000 0X0000
% B9:180 % 0X0000 0X0000 0X0000 0X0000 0X0000 0X0002 0X0000 0X0000 0X0000 0X0000
% B9:190 % 0X0010 0X0000 0X0000 0X0000 0X0000 0X0000 0X0000 0X0000 0X0000 0X0000
% B9:200 % 0X2B64 0X2B64 0X0000 0X0010 0X0000 0X2000 0X0000 0X0000 0X0000 0X0000
% B9:220 % 0X0000 0X0000 0X0000 0X0200 0X0000 0X0000 0X0000 0X0000 0X0000 0X0020
% B9:230 % 0X0040 0X0000 0X0000 0X0000 0X0000 0X0000 0X0000 0X0000 0X0000 0X0000
DATA B11
% B11:180 % 0X0000 0X8000 0X0000 0X0000 0X0000 0X0000 0X0000 0X0000 0X0000 0X0000
% B11:240 % 0X0000 0X0000 0X0000 0X4000 0X0000 0X0000 0X0000 0X0000 0X0000 0X0000
DATA B12
% B12:0 % 0X0068 0X0000 0X0000 0X0000 0X0000 0X0000 0X0000 0X0000 0X0000 0X0000
DATA L13
% L13:0 % 4994 5000 6 300 -1207775130
% L13:5 % 4 3 4 176627 341852
% L13:10 % 0 3 0 0 333
% L13:15 % 7535567 -2147483648 2147483647 0 1867350
% L13:20 % -1974778253 6884924 500 37037 0
% L13:25 % 1400 32 36 35 8
% L13:30 % -1975106214 0 32 23 0
% L13:35 % 1867 0 -1975106214 0 46
% L13:40 % 0 0 100 20 0
% L13:45 % 26 0 128 78459887 -1207775104
% L13:50 % 111480 1950650196 6278 0 5000
% L13:55 % 26 14 26 1950650196 666
% L13:60 % 0 227 11148000 49110 7
% L13:65 % 26 5 -1477234292 5 6884956
% L13:70 % -1477186136 -1477186176 40 5 5
% L13:75 % 104209 213 1619 4357 99
% L13:80 % 29 411541266 150 0 999999
% L13:85 % 12 200 45 26483 1000
% L13:90 % 26616 0 54 1000 0
% L13:95 % 60 99000 99000 25989 99000
% L13:100 % -1478910248 1 26 43 2025
% L13:105 % 1 0 -1975106318 18668 -1975106326
% L13:110 % 8 30 15 537159595 537159593
% L13:115 % 537159600 7 4 537159596 1
% L13:120 % 0 50 0 30 49
% L13:125 % 164 19 155494060 137 155494060
% L13:130 % 1 1 0 2 0
% L13:135 % 0 1000 111 12 0
% L13:140 % 0 11 12 0 20
% L13:145 % 2568 1273 1284 111 111
% L13:150 % -1538760531 -1538760111 88 0 100
% L13:155 % 420 332 24 0 262301
% L13:160 % 3 7 4 395082 53203921
% L13:165 % 3 189116 95 13 8150
% L13:170 % 55946610 53 72 54 13
% L13:175 % 0 0 42 23 2021
% L13:180 % 176247033 25 99000 52866 644409
% L13:185 % 64 916459 92 627156 63
% L13:190 % 4 5 666 650831 0
DATA F14
% F14:0 % 0 0 0 76 0
DATA N15
% N15:0 % 0 0 0 0 0 108 0 1310 0 10
DATA L16
% L16:0 % 8 14 11 0 20
% L16:5 % 250 5000 5000 182 19
% L16:10 % 1256 18 2045 6599584 98
% L16:15 % 99 0 0 0 0
DATA B17
% B17:60 % 0XC000 0X0000 0X0000 0X0000 0X0000 0X0000 0X0000 0X0000 0X0000 0X0000
% B17:100 % 0X0000 0X0000 0X0000 0X0000 0X0000 0X0000 0X0000 0X0000 0X1000 0X0000
% B17:110 % 0X4000 0X0000 0X0000 0X0000 0X0000 0X0000 0X0000 0X0000 0X0000 0X0000
% B17:120 % 0X0000 0X0000 0X0000 0X0000 0X0000 0X0000 0X0000 0X2000
DATA B18
% B18:60 % 0XC000 0X0000 0X0000 0X0000 0X0000 0X0000 0X0000 0X0000 0X0000 0X0000
% B18:100 % 0X0000 0X0000 0X0000 0X0000 0X0000 0X0000 0X0000 0X0000 0X0000 0X8240
% B18:110 % 0X0000 0X0400 0X0000 0X0000 0X0000 0X0000 0X0040 0X0000 0X0000 0X0010
% B18:120 % 0X0000 0X0000 0X0000 0X0000 0X0000 0X0000 0X0000 0X2000
DATA L23
% L23:0 % 65535 -65536 -65536 -65536 -65536
% L23:5 % -65536 -65536 2 65535 -65536
% L23:10 % -65536 0 17 10 17
% L23:15 % 0 0 0 0 8
% L23:20 % 0 -65536 -65536 -65536 -65536
% L23:25 % -65536 20 19 20 0
% L23:30 % 0 0 -65536 -65536 -65536
% L23:35 % -65536 -65536 -65536 -65536 -65536
% L23:40 % 16270 18414 0 63266 -65536
% L23:45 % 5062 0 0 0 0
% L23:50 % 0 -65536 -65536 17 -65536
% L23:55 % 33 5079 -65536 0 0
% L23:60 % 0 -65536 -65536 -65536 0
DATA L24
% L24:0 % -65536 122 -65536 222 -65536
% L24:5 % 65535 -65536 -65536 -65536 -65536
% L24:10 % 50 27 0 1 23
% L24:15 % 1198 1030 95 18 30
% L24:20 % 30 -65536 1226 -65536 -65536
% L24:25 % 222 1236 -65536 -65536 222
% L24:30 % 1466 27 10000 -65536 55
% L24:35 % 180 -65536 180 65535 101
% L24:40 % 101 1000 -65536 -65536 10
% L24:45 % 222 192 -65536 0 -65536
% L24:50 % -999 30 10000 65535 900
DATA L27
% L27:0 % -734752198 -734752002 -734751806 -734751581 -734751403
% L27:5 % -734751201 -734750999 -734750792 -734750579 -734750387
% L27:10 % -734750268 -734750086 -734749985 -726361081 -734749480
% L27:15 % -734749286 -734749075 -734748974 -734748775 -734748551
% L27:20 % -734748367 -734748168 -734747969 -734747774 -734747667
% L27:25 % -734747437 -734747264 -734747138 -734746858 -734746760
% L27:30 % -734746539 -734746363 -734746161 -734746054 -734745859
% L27:35 % -734745651 -734745455 -734745341 -734745129 -734744925
% L27:40 % -734744744 -734744527 -734744324 -734744138 -734743944
% L27:45 % -734743829 -734743635 -734743407 -734743232 -734743036
DATA L28
% L28:0 % 6475838 6475903 6475961 6476018 6476075
% L28:5 % 6476129 6476191 6476246 6476309 6476365
% L28:10 % 6476426 6476482 6476548 6476601 6476660
% L28:15 % 6476713 6476775 6476834 6476894 6476960
% L28:20 % 6477012 6477081 6477138 6630544 6721998
% L28:25 % 6818212 6831084 6847887 6884924 6474577
% L28:30 % 6474650 6474729 6474789 6474851 6474911
% L28:35 % 6474965 6475030 6475088 6475141 6475200
% L28:40 % 6475257 6475309 6475379 6475436 6475495
% L28:45 % 6475554 6475613 6475666 6475722 6475780
DATA L29
% L29:0 % -1975312412 -1975312379 -1975312350 -1975312321 -1975312292
% L29:5 % -1975312265 -1975312234 -1975312206 -1975312174 -1975312146
% L29:10 % -1975312115 -1975312087 -1975312054 -1975312027 -1975311997
% L29:15 % -1975311970 -1975311939 -1975311909 -1975311879 -1975311846
% L29:20 % -1975311820 -1975311785 -1975311756 -1975234431 -1975188339
% L29:25 % -1975139843 -1975133354 -1975124882 -1975106214 -1975313047
% L29:30 % -1975313010 -1975312970 -1975312940 -1975312909 -1975312879
% L29:35 % -1975312852 -1975312819 -1975312790 -1975312763 -1975312733
% L29:40 % -1975312704 -1975312678 -1975312643 -1975312615 -1975312585
% L29:45 % -1975312555 -1975312525 -1975312498 -1975312470 -1975312441
DATA L30
% L30:0 % -1283861654 -1283860474 -1283858758 -1283845411 -1283844812
% L30:5 % -1283843877 -1283841466 -1283839546 -1283838837 -1283834821
% L30:10 % -1283833088 -1283829339 -1283829122 -1283824619 -1283822332
% L30:15 % -1283815346 -1283814532 -1283813200 -1283809112 -1283802804
% L30:20 % -1283797988 -1283786341 -1283760626 -1283744192 -1283717906
% L30:25 % -1283696915 -1207777165 -1207776938 -1207775584 -1207775357
% L30:30 % -1207775130 -1283942245 -1283941742 -1283941489 -1283940982
% L30:35 % -1283940127 -1283939882 -1283939142 -1283937555 -1283937231
% L30:40 % -1283936439 -1283936163 -1283935127 -1283934876 -1283933278
% L30:45 % -1283877537 -1283875223 -1283873897 -1283870637 -1283861929
DATA L31
% L31:0 % 1921863169 1921863763 1921864627 1921871355 1921871657
% L31:5 % 1921872129 1921873343 1921874311 1921874669 1921876692
% L31:10 % 1921877566 1921879456 1921879565 1921881835 1921882987
% L31:15 % 1921886508 1921886919 1921887591 1921889651 1921892831
% L31:20 % -225588390 1921901129 1921914091 1921922373 1921935623
% L31:25 % 1921946202 1950650196 1950650196 1950650196 1950650196
% L31:30 % 1950650196 1921822553 1921822806 1921822934 1921823189
% L31:35 % 1921823620 1921823744 1921824117 1921824917 1921825080
% L31:40 % 1921825478 1921825617 1921826139 1921826265 1921827071
% L31:45 % 1921855164 1921856330 1921857000 1921858641 1921863030
DATA L42
% L42:0 % -2042345216 -734706020 -734705920 -734705705 -734705537
% L42:5 % -734705422 -734705217 -734704927 -734704823 -734704618
% L42:10 % -734704423 -734704314 -734704102 -734703886 -734703717
% L42:15 % -734703510 -734703412 -734703170 -734703007 -734702810
% L42:20 % -734702606 -734702492 -734702194 -734702010 -734701798
% L42:25 % -734701700 -734701496 -734701395 -734701181 -734700895
% L42:30 % -734700788 -734700590 -734700390 -734700289 -734699993
% L42:35 % -734699874 -734699685 -734699489 -734699379 -734699164
% L42:40 % -734698976 -734698778 -734698574 -734698375 -734698164
% L42:45 % -734697977 -734697767 -734697574 -734697464 -734697264
% L42:50 % -734697150 -734696959
DATA B181
% B181:0 % 0X6AC0 0XD435 0X6B2C 0XD435 0X6BF9 0XD435 0X6C64 0XD435 0X6D3D 0XD435
% B181:10 % 0X6DFA 0XD435 0X6EBB 0XD435 0X6F80 0XD435 0X704E 0XD435 0X7118 0XD435
% B181:20 % 0X71D7 0XD435 0X72A0 0XD435 0X730C 0XD435 0X737E 0XD435 0X749F 0XD435
% B181:30 % 0X7584 0XD435 0X764A 0XD435 0X76F5 0XD435 0X777A 0XD435 0X782B 0XD435
% B181:40 % 0X795A 0XD435 0X79C4 0XD435 0X12B5 0XD434 0X1371 0XD434 0X1437 0XD434
% B181:50 % 0X14FF 0XD434 0X157F 0XD434 0X1632 0XD434 0X1755 0XD434 0X181D 0XD434
% B181:60 % 0X188E 0XD434 0X195A 0XD434 0X1A1E 0XD434 0X1B02 0XD434 0X1BD2 0XD434
% B181:70 % 0X1C8E 0XD434 0X1D3C 0XD434 0X1E06 0XD434 0X1ED6 0XD434 0X1F4E 0XD434
% B181:80 % 0X2005 0XD434 0X20C7 0XD434 0X2197 0XD434 0X2276 0XD434 0X2331 0XD434
% B181:90 % 0X23EE 0XD434 0X24B9 0XD434 0X2526 0XD434 0X25E6 0XD434 0X26D2 0XD434
% B181:100 % 0X277A 0XD434 0X284A 0XD434 0X2917 0XD434 0X297B 0XD434 0X2A54 0XD434
% B181:110 % 0X2B1D 0XD434 0X2BD7 0XD434 0X2C98 0XD434 0X2D05 0XD434 0X2DCE 0XD434
% B181:120 % 0X2E90 0XD434 0X2F62 0XD434 0X2FCA 0XD434 0X3092 0XD434 0X3157 0XD434
% B181:130 % 0X3224 0XD434 0X32E4 0XD434 0X3351 0XD434 0X33C8 0XD434 0X3485 0XD434
% B181:140 % 0X3541 0XD434 0X361F 0XD434 0X36DF 0XD434 0X379F 0XD434 0X3870 0XD434
% B181:150 % 0X3937 0XD434 0X39A5 0XD434 0X3A72 0XD434 0X3B29 0XD434 0X3BFB 0XD434
% B181:160 % 0X3C72 0XD434 0X3D2A 0XD434 0X3E1A 0XD434 0X3EBF 0XD434 0X3F84 0XD434
% B181:170 % 0X4001 0XD434 0X411A 0XD434 0X41F7 0XD434 0X42A4 0XD434 0X431A 0XD434
% B181:180 % 0X43D2 0XD434 0X4454 0XD434 0X450E 0XD434 0X45E1 0XD434 0X46A1 0XD434
% B181:190 % 0X476D 0XD434 0X488D 0XD434 0X4956 0XD434 0X4A27 0XD434 0X4AA1 0XD434
% B181:200 % 0X4B58 0XD434 0X4C1E 0XD434 0X4CA0 0XD434 0X4DBB 0XD434 0X4E22 0XD434
% B181:210 % 0X4ED9 0XD434 0X4F51 0XD434 0X5008 0XD434 0X50D1 0XD434 0X513E 0XD434
% B181:220 % 0X526E 0XD434 0X52D1 0XD434 0X53B6 0XD434 0X545D 0XD434 0X54D0 0XD434
% B181:230 % 0X55A2 0XD434 0X565F 0XD434 0X571E 0XD434 0X578E 0XD434 0X584D 0XD434
% B181:240 % 0X5916 0XD434 0X59E0 0XD434 0X5A61 0XD434 0X5B73 0XD434 0X5BEE 0XD434
% B181:250 % 0X5CB2 0XD434 0X5DF6 0XD434 0X5E9B 0XD434
DATA F182
% F182:0 % -3.098753e+12 -3.098806e+12 -3.098859e+12 -3.098886e+12 -3.098942e+12
% F182:5 % -3.098991e+12 -3.099044e+12 -3.09907e+12 -3.099103e+12 -3.099201e+12
% F182:10 % -3.099231e+12 -3.099284e+12 -3.099335e+12 -3.099386e+12 -3.099445e+12
% F182:15 % -3.099494e+12 -3.099546e+12 -3.099599e+12 -3.099652e+12 -3.099707e+12
% F182:20 % -3.099732e+12 -3.099784e+12 -3.099837e+12 -3.099864e+12 -3.099914e+12
% F182:25 % -3.099974e+12 -3.100025e+12 -3.100075e+12 -3.100125e+12 -3.100159e+12
% F182:30 % -3.100207e+12 -3.100267e+12 -3.100318e+12 -3.100365e+12 -3.100416e+12
% F182:35 % -3.100445e+12 -3.1005e+12 -3.10055e+12 -3.100603e+12 -3.100654e+12
% F182:40 % -3.10069e+12 -3.100736e+12 -3.100786e+12 -3.100839e+12 -3.100868e+12
% F182:45 % -3.100921e+12 -3.100973e+12 -3.10105e+12 -3.101079e+12 -3.105427e+12
DATA L183
% L183:0 % -734756123 -734755929 -734755729 -734755497 -734755333
% L183:5 % -734755123 -734755023 -734754817 -734754602 -734754419
% L183:10 % -734754215 -734754024 -717976671 -734753716 -734753501
% L183:15 % -734753306 -734753106 -734752915 -734752801 -734752594
% L183:20 % -734752411 0 0 0 0
DATA B185
% B185:0 % 0X0200 0X0001 0X0000 0X0000 0X0000 0X0000 0X2000 0X0000 0X0000 0X0000
DATA N186
% N186:0 % 100 0 0 0 0 0 0 0 0 0
DATA L187
% L187:0 % 34 26 497 0 524288
DATA F188
% F188:0 % 0 66 11 44 29
DATA B189
% B189:0 % 0X00F1 0X0000 0X0000 0X0000 0X0000 0X0000 0X0000 0X0000 0X0000 0X0000
DATA L190
% L190:0 % 1 5 0 0 0
% L190:30 % 0 2 0 0 0
% L190:35 % -2145386496 256 0 0 0
DATA B191
% B191:0 % 0X0000 0X0001 0X0000 0X0000 0X0000 0X0000 0X0000 0X0000 0X0000 0X0000
DATA L192
% L192:0 % -1476963844 266932201 5055 81 0
% L192:5 % 1000000 253000000 999 999 8
% L192:10 % 0 0 2097153 78 17
% L192:15 % -1444152439 332250347 860888 77 0
% L192:20 % 180 39200000 0 0 0
DATA F193
% F193:0 % 0.3903424 0.315 0.022 6 0
% F193:5 % 0 0.02 0 0 419.7934
% F193:10 % 0.011 0.195 0.165 0.337 760
% F193:15 % -0.3382568 0.25 -0.08456421 696.6768 22827.31
DATA B194
% B194:120 % 0X0000 0X0000 0X0000 0X0000 0X0000 0X0000 0X0000 0X8000
DATA B195
% B195:90 % 0X0000 0X0000 0X0000 0X0000 0X0000 0X0000 0X0000 0X0040 0X0000 0X0000
DATA B196
% B196:0 % 0X0E26 0X9FF4 0X0005 0X0000 0X0000 0X0000 0X0000 0X0000 0X0000 0X0000
% B196:30 % 0XE800 0X9BFF 0XEBFF 0XFFDF 0XFFFF 0X0000 0X0000 0X0000 0X0000 0X0000
DATA N197
% N197:0 % 1560 150 500 2500 2500 14417 5555 0 200 0
% N197:10 % 4000 969 4 0 0 0 0 0 0 0
% N197:30 % 15 48 0 0 0 0 0 0 0 0
DATA B198
% B198:0 % 0X0009 0X0000 0X0000 0X0000 0X0000 0X0000 0X0000 0X0000 0X0000 0X0000
DATA L199
% L199:0 % 1 5571998 134 11 3579521
% L199:5 % 0 0 0 5 1064359
% L199:10 % 0 224 10256 556 0
% L199:15 % 0 0 0 278717848 518
% L199:20 % 28295 16430853 5001 5001 0
% L199:25 % 0 0 28329 1 3781224
% L199:30 % 21630086 251 3809367 15030467 111
% L199:35 % 555 555 0 0 0
DATA N200
% N200:0 % 2046 124 1 2047 1172 1594 1004 2045 2045 2045
% N200:10 % 0 0 0 1277 178 2046 1000 2045 2045 1218
% N200:20 % 1555 0 0 0 0 0 0 0 0 0
% N200:30 % 0 0 32767 0 0 0 0 0 0 0
DATA L201
% L201:0 % 20 40 40 -3011735 44
% L201:5 % 96629277 0 0 -3010662 0
% L201:10 % 0 0 0 327 43
% L201:15 % 0 43 0 43 36830
DATA B202
% B202:0 % 0X2241 0X0000 0X0001 0X0000 0X0000 0X0000 0X0000 0X0000 0X0000 0X0000
DATA N203
% N203:0 % 115 115 116 333 334 333 444 0 445 444
% N203:10 % 555 556 555 0 0 0 0 0 0 0
DATA L204
% L204:0 % 333 0 333 1362 124
% L204:5 % 2000 2000 462 222 0
% L204:10 % 0 0 0 1327077052 1327077052
% L204:15 % 1327077052 1327077052 1 0 0
% L204:20 % 0 0 33 0 0
% L204:30 % 33 0 0 0 0
DATA F205
% F205:0 % 25 66 0 66 0
